// TIA Portal V18 export
VAR_GLOBAL   // PLC tag table "S1_R1"
   S1_R1_Valve_Up AT %Q300.0 : Bool;
   S1_R1_Valve_Down AT %Q300.1 : Bool;
   S1_R1_Sen_Drv_1 AT %I300.0 : Bool;
   S1_R1_Sen_Drv_2 AT %I300.1 : Bool;
   S1_R1_Sen_Drv_3 AT %I300.2 : Bool;
   S1_R1_Sen_Drv_4 AT %I300.3 : Bool;
   S1_R1_Sen_Val1_Up AT %I300.4 : Bool;
   S1_R1_Sen_Val1_Down AT %I300.5 : Bool;
   S1_R1_Sen_Val2_Up AT %I300.6 : Bool;
   S1_R1_Sen_Val2_Down AT %I300.7 : Bool;
   S1_R1_Hyd_Filtr AT %I301.0 : Bool;
   S1_R1_Hyd_Empty AT %I301.1 : Bool;
   S1_R1_Safety1_1 AT %I350.0 : Bool;
   S1_R1_Safety2_1 AT %I350.1 : Bool;
   S1_R1_Safety3_1 AT %I350.2 : Bool;
   S1_R1_Safety4_1 AT %I350.3 : Bool;
   S1_R1_Safety1_2 AT %I351.0 : Bool;
   S1_R1_Safety2_2 AT %I351.1 : Bool;
   S1_R1_Safety3_2 AT %I351.2 : Bool;
   S1_R1_Safety4_2 AT %I351.3 : Bool;
END_VAR
